FUNCTION_BLOCK FB_IODEV_CHANNEL
VAR_INPUT
END_VAR
VAR_OUTPUT
END_VAR
VAR
END_VAR

METHOD M_Compute
VAR_INPUT
END_VAR
END_METHOD

METHOD M_Reset
VAR_INPUT
END_VAR
END_METHOD

END_FUNCTION_BLOCK

(* stored: Version 1.1.0.1, ProductVersion 3.1.4022.9
   POU FB_IODEV_CHANNEL: Id {5cd2f090-79d0-4419-8b4e-39862b4bf3b7}, SpecialFunc None
   Method M_Compute: Id {d883c9b0-499e-41da-af16-322def6b3a9d}
   Method M_Reset: Id {92348419-62cc-4cb8-8025-79fcbbae164f} *)
